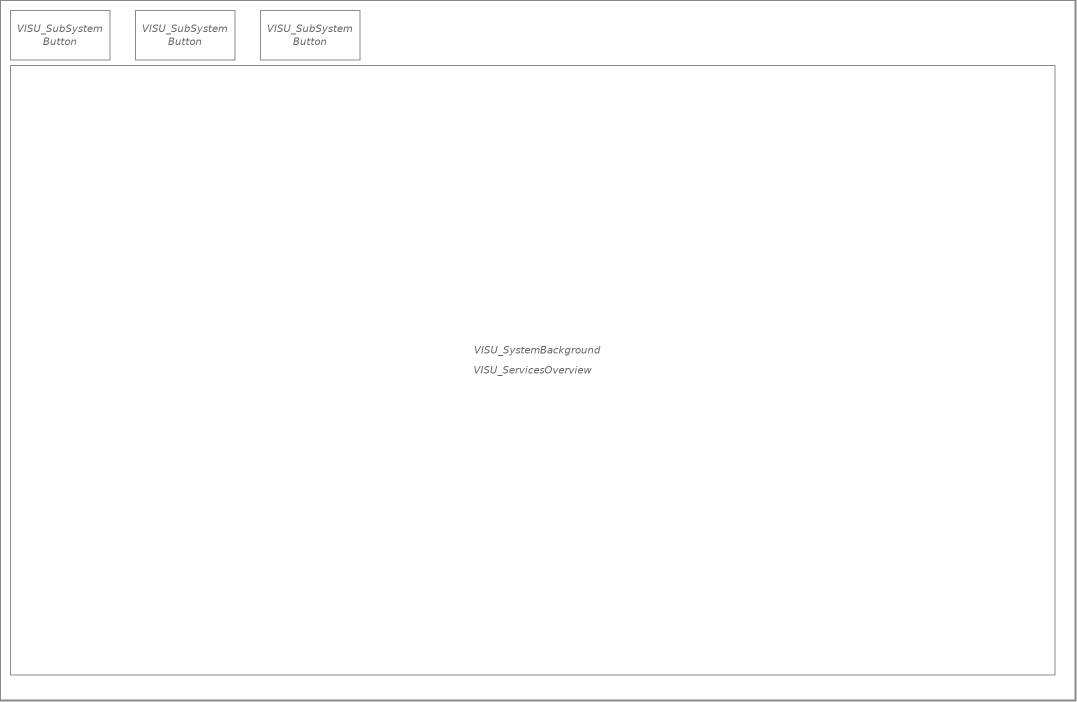
VISUALIZATION VISU_Services  // 1077x702
VAR_IN_OUT
	ref : Services;
    widget : ServicesWidget;
END_VAR
    Frame (0,0 1075x700)
        shows VISU_SystemBackground(color := widget.actualStatus.color)
    Frame (10,65 1045x610)
        shows VISU_ServicesOverview(ref := ref, widget := widget)
        shows VISU_ServicesTiming(ref := ref.parts.timing, widget := widget.timing)
        shows VISU_ServicesConfig(editableConfig := ref.editableConfig, activeConfig := ref.config, mgr := ref.parts.configManager, mgrWidget := widget.configManager, activeTab := widget.configActiveTab)
    Frame (10,10 100x50)
        shows VISU_SubSystemButton(widget := widget.button_overview)
        OnMouseClick: FrameSelectionChange Selection=SelectedFrame=b1e9e4b0-bf3d-440f-90c5-cb513105ccf1, GlobSel=AssignType=Directly, SelType=Locally
        OnMouseClick: execute { widget.activeTab := ServicesTabs.OVERVIEW; }
    Frame (135,10 100x50)
        shows VISU_SubSystemButton(widget := widget.button_timing)
        OnMouseClick: FrameSelectionChange Selection=SelectedFrame=b1e9e4b0-bf3d-440f-90c5-cb513105ccf1, Selection=1, GlobSel=AssignType=Directly, SelType=Locally
        OnMouseClick: execute { widget.activeTab := ServicesTabs.TIMING; }
    Frame (260,10 100x50)
        shows VISU_SubSystemButton(widget := widget.button_config)
        OnMouseClick: FrameSelectionChange Selection=SelectedFrame=b1e9e4b0-bf3d-440f-90c5-cb513105ccf1, Selection=2, GlobSel=AssignType=Directly, SelType=Locally
        OnMouseClick: execute { widget.activeTab := ServicesTabs.CONFIG; }
END_VISUALIZATION

(* stored: Version 1.1.0.1, ProductVersion 3.1.4019.2
   Visu VISU_Services: Id {c32e5802-8e40-41cc-9eb8-ab40fb98def0} *)
